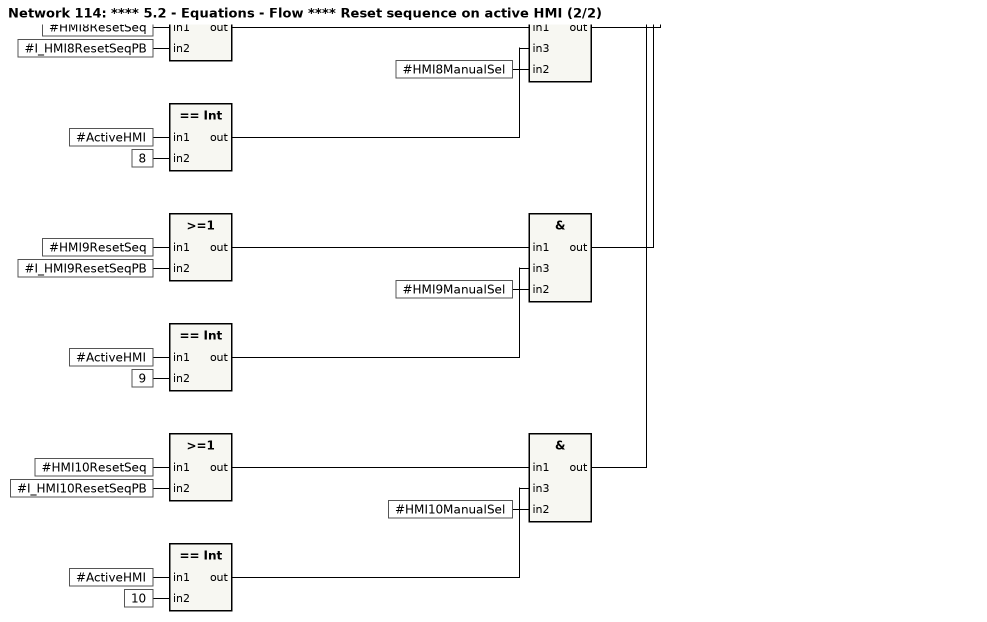
   #O_ResetSeqSel := ((#HMI1ResetSeq OR #I_HMI1ResetSeqPB) AND (#ActiveHMI = 1) AND #HMI1ManualSel) OR ((#HMI2ResetSeq OR #I_HMI2ResetSeqPB) AND (#ActiveHMI = 2) AND #HMI2ManualSel) OR ((#HMI3ResetSeq OR #I_HMI3ResetSeqPB) AND (#ActiveHMI = 3) AND #HMI3ManualSel) OR ((#HMI4ResetSeq OR #I_HMI4ResetSeqPB) AND (#ActiveHMI = 4) AND #HMI4ManualSel) OR ((#HMI5ResetSeq OR #I_HMI5ResetSeqPB) AND (#ActiveHMI = 5) AND #HMI5ManualSel) OR ((#HMI6ResetSeq OR #I_HMI6ResetSeqPB) AND (#ActiveHMI = 6) AND #HMI6ManualSel) OR ((#HMI7ResetSeq OR #I_HMI7ResetSeqPB) AND (#ActiveHMI = 7) AND #HMI7ManualSel) OR ((#HMI8ResetSeq OR #I_HMI8ResetSeqPB) AND (#ActiveHMI = 8) AND #HMI8ManualSel) OR ((#HMI9ResetSeq OR #I_HMI9ResetSeqPB) AND (#ActiveHMI = 9) AND #HMI9ManualSel) OR ((#HMI10ResetSeq OR #I_HMI10ResetSeqPB) AND (#ActiveHMI = 10) AND #HMI10ManualSel);
   #IO_Modes.LModeSelector.ResetSeqSel := #O_ResetSeqSel;
END_REGION

REGION Network 115: **** 5.2 - Equations - Flow **** Check Active HMI again - HMI <> 0
   // Check Active HMI again
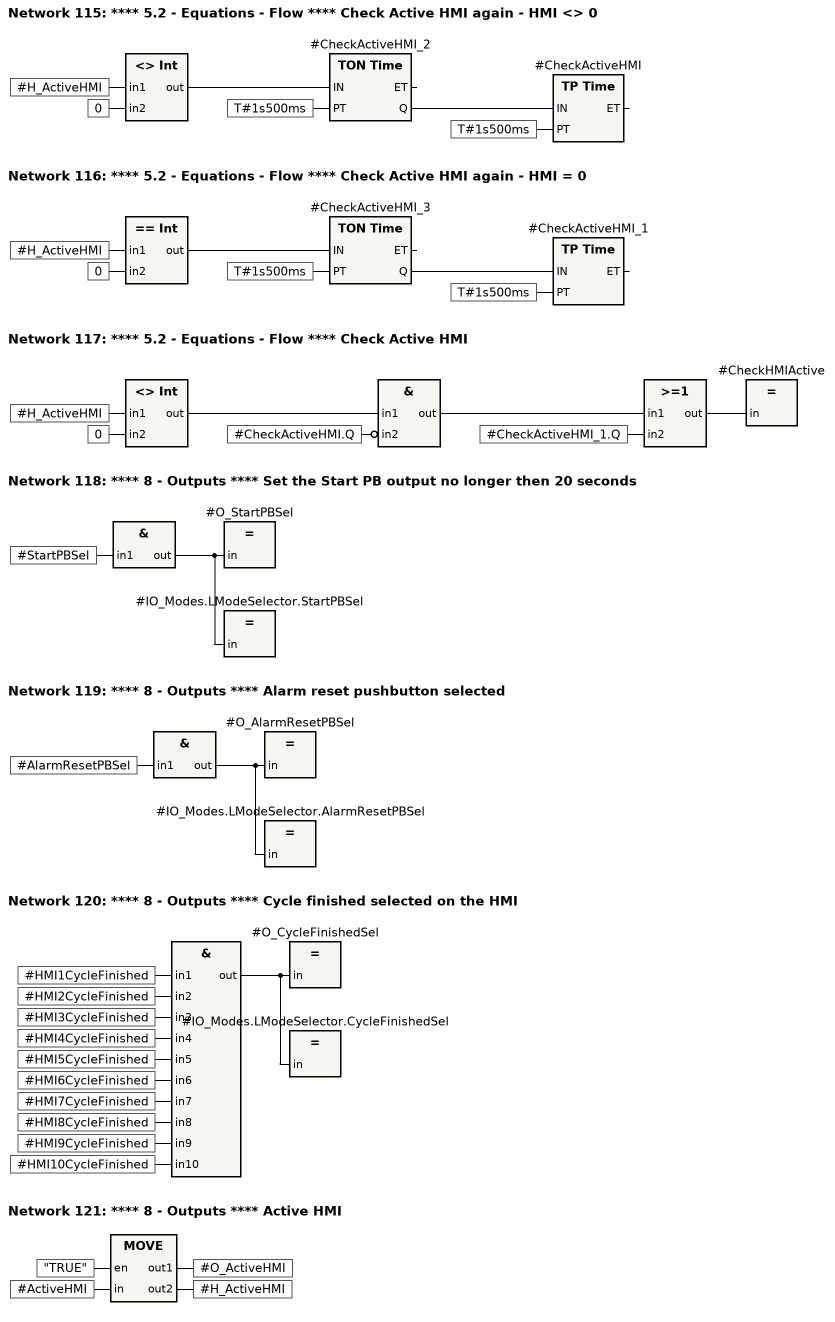
   #CheckActiveHMI_2(IN := #H_ActiveHMI <> 0, PT := T#1s500ms);   // TON
   #CheckActiveHMI(IN := #CheckActiveHMI_2.Q, PT := T#1s500ms);   // TP
END_REGION

REGION Network 116: **** 5.2 - Equations - Flow **** Check Active HMI again - HMI = 0
   // Check Active HMI again
   #CheckActiveHMI_3(IN := #H_ActiveHMI = 0, PT := T#1s500ms);   // TON
   #CheckActiveHMI_1(IN := #CheckActiveHMI_3.Q, PT := T#1s500ms);   // TP
END_REGION

REGION Network 117: **** 5.2 - Equations - Flow **** Check Active HMI
   // Check Active HMI
   #CheckHMIActive := ((#H_ActiveHMI <> 0) AND NOT #CheckActiveHMI.Q) OR #CheckActiveHMI_1.Q;
END_REGION

REGION Network 118: **** 8 - Outputs **** Set the Start PB output no longer then 20 seconds
   // Set the Start PB output no longer then 20 seconds
   #O_StartPBSel := #StartPBSel;
   #IO_Modes.LModeSelector.StartPBSel := #StartPBSel;
END_REGION

REGION Network 119: **** 8 - Outputs **** Alarm reset pushbutton selected
   // Alarm reset pushbutton selected
   #O_AlarmResetPBSel := #AlarmResetPBSel;
   #IO_Modes.LModeSelector.AlarmResetPBSel := #AlarmResetPBSel;
END_REGION

REGION Network 120: **** 8 - Outputs **** Cycle finished selected on the HMI
   // Cycle finished selected on the HMI
   #O_CycleFinishedSel := #HMI1CycleFinished AND #HMI2CycleFinished AND #HMI3CycleFinished AND #HMI4CycleFinished AND #HMI5CycleFinished AND #HMI6CycleFinished AND #HMI7CycleFinished AND #HMI8CycleFinished AND #HMI9CycleFinished AND #HMI10CycleFinished;
   #IO_Modes.LModeSelector.CycleFinishedSel := #O_CycleFinishedSel;
END_REGION

REGION Network 121: **** 8 - Outputs **** Active HMI
   // Active HMI
   IF "TRUE" THEN
       #O_ActiveHMI := #ActiveHMI;
       #H_ActiveHMI := #ActiveHMI;
   END_IF;
END_REGION

REGION Network 122: **** 8 - Outputs **** Lock Manual Time
   // Lock Manual Time
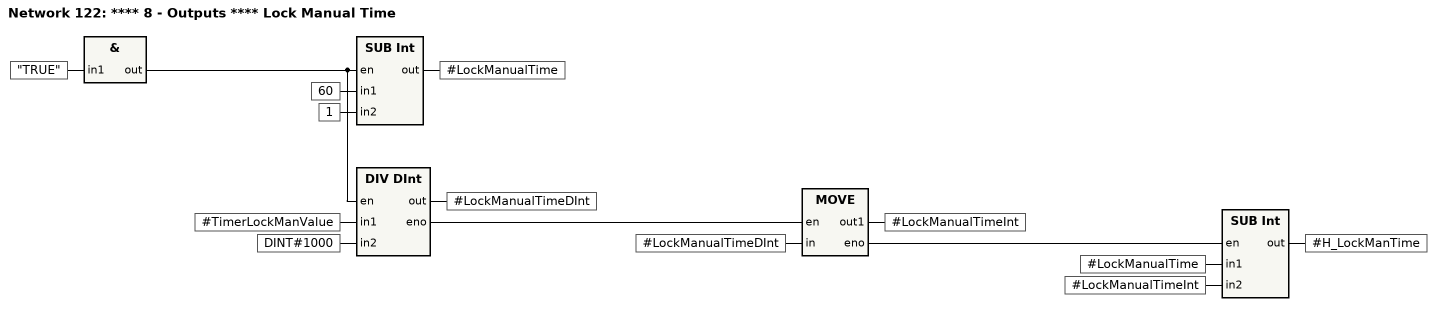
   // ENO of a box is taken as its EN; it also drops when the box reports an error
   IF "TRUE" THEN
       #LockManualTime := 60 - 1;
       #LockManualTimeDInt := #TimerLockManValue / DINT#1000;
       #LockManualTimeInt := #LockManualTimeDInt;
       #H_LockManTime := #LockManualTime - #LockManualTimeInt;
   END_IF;
END_REGION
END_FUNCTION_BLOCK
